Staubli VAL3: Blend.pjx

--- Blend.pjx ---
Parameters version=s7.9 stackSize=5000 millimeterUnit=true
Program file=Carterblend.pgx
Program file=JointBlend.pgx
Program file=start.pgx
Program file=stop.pgx
Data file=Blend.dtx

--- Carterblend.pgx ---
program Carterblend()
begin

  //直线与圆弧



  //直线与直线




  //圆弧与直线



  //圆弧与圆弧














end
